// TIA Portal V17 export
// export: Created 2023-04-06T14:59:51.4519566Z, ExportSetting None, DisplayName Totally Integrated Automation Portal, DisplayVersion V17 Update 4, DisplayName TIA Portal Openness, DisplayVersion V17 Update 4, DisplayName TIA Portal Version Control Interface, DisplayVersion V17, DisplayName STEP 7 Professional, DisplayVersion V17 Update 4, DisplayName STEP 7 Safety, DisplayVersion V17, DisplayName WinCC Advanced / Unified PC, DisplayVersion V17 Update 4
DATA_BLOCK "SETTINGS"   // DB26
{ S7_Optimized_Access := 'FALSE' }
// stored: AutoNumber false
   VAR RETAIN
      LT_500 : Struct   // AI 5
         RANGE_L : Real := 70.0;
         RANGE_H : Real := 80.0;
         SP_LL : Real := -30.0;
         SP_L : Real := -30.0;
         SP_H : Real := 180.0;
         SP_HH : Real := 180.0;
      END_STRUCT;
      VT_600 : Struct   // AI 6
         RANGE_L : Real := -80.0;
         RANGE_H : Real := -40.0;
         SP_LL : Real := -180.0;
         SP_L : Real := -180.0;
         SP_H : Real := 60.0;
         SP_HH : Real := 60.0;
      END_STRUCT;
      PT_200 : Struct   // AI 2
         RANGE_L : Real := -10.0;
         RANGE_H : Real := 20.0;
         SP_LL : Real := -110.0;
         SP_L : Real := -110.0;
         SP_H : Real := 120.0;
         SP_HH : Real := 120.0;
      END_STRUCT;
      FT_400 : Struct   // AI 4
         RANGE_L : Real := 20.0;
         RANGE_H : Real := 60.0;
         SP_LL : Real := -80.0;
         SP_L : Real := -80.0;
         SP_H : Real := 160.0;
         SP_HH : Real := 160.0;
      END_STRUCT;
      PT_100 : Struct   // AI 1
         RANGE_L : Real := 0.0;
         RANGE_H : Real := 100.0;
         SP_LL : Real := -100.0;
         SP_L : Real := -100.0;
         SP_H : Real := 200.0;
         SP_HH : Real := 200.0;
      END_STRUCT;
      TT_300 : Struct   // AI 3
         RANGE_L : Real := -30.0;
         RANGE_H : Real := 512.0;
         SP_LL : Real := -130.0;
         SP_L : Real := -130.0;
         SP_H : Real := 612.0;
         SP_HH : Real := 612.0;
      END_STRUCT;
   END_VAR
BEGIN
END_DATA_BLOCK
